FUNCTION_BLOCK FB_Station IMPLEMENTS I_Station
VAR
	refCylinder	: REFERENCE TO FB_Cylinder;
	_eState		: E_StationState;
	_eCommand	: E_Command;
	_stStatus	: ST_StationStatus;
	_stRecipe	: ST_Recipe;
	_uWord		: U_Word;
	_sIdent		: T_Ident;
	_nErrorId	: UDINT;
END_VAR

Cyclic();

METHOD Cyclic
VAR
	bExtended	: BOOL;
END_VAR
bExtended := refCylinder.bIsExtended;

CASE _eState OF
	E_StationState.Idle:
		IF _eCommand = E_Command.Start THEN
			_eState := E_StationState.Running;
		END_IF

	E_StationState.Running:
		IF bExtended THEN
			refCylinder.Retract();
		ELSE
			refCylinder.Extend();
		END_IF
		IF _nErrorId <> 0 THEN
			_eState := E_StationState.Error;
		END_IF

	E_StationState.Error:
		_stStatus.bError := TRUE;

	E_StationState.Done:
		_stStatus.bDone := TRUE;
END_CASE

_stStatus.eState := _eState;
_stStatus.nErrorId := _nErrorId;
_uWord.nWord := _stRecipe.aSteps[1];
END_METHOD

METHOD Execute : BOOL
VAR
END_VAR
IF _eState = E_StationState.Idle THEN
	_eCommand := E_Command.Start;
	_stStatus.bBusy := TRUE;
	Execute := TRUE;
ELSE
	Execute := FALSE;
END_IF
END_METHOD

METHOD Reset : BOOL
VAR
END_VAR
_eState := E_StationState.Idle;
_eCommand := E_Command.None;
_nErrorId := 0;
_stStatus.bBusy := FALSE;
_stStatus.bDone := FALSE;
_stStatus.bError := FALSE;
_stStatus.nErrorId := 0;
Reset := TRUE;
END_METHOD

PROPERTY State : E_StationState
GET
State := _eState;
END_GET
SET
_eState := State;
END_SET
END_PROPERTY

PROPERTY ErrorId : UDINT
GET
ErrorId := _nErrorId;
END_GET
END_PROPERTY

ACTION Act_Home:
refCylinder REF= GVL_System.fbCylinder;
refCylinder.Retract();
_eState := E_StationState.Idle;
_sIdent := 'STATION-01';
END_ACTION

END_FUNCTION_BLOCK

(* stored: Version 1.1.0.1, ProductVersion 3.1.4024.12
   POU FB_Station: Id {ba9b86f0-e4ae-49bd-8d10-d23550802ca5}, SpecialFunc None
   Folder Actions: Id {e81da3d1-8551-49cc-bce9-534df56315e3}
   Method Cyclic: Id {d83d5f63-b782-429a-b4e4-1fd8aac79cdb}
   Method Execute: Id {e043de6a-b3b7-4a09-ac5a-903c66262592}
   Method Reset: Id {ed197d53-3022-4f16-b73a-835f98c1ee8e}
   Property State: Id {0eea66ef-e1f3-405c-94a3-a03642077656}
   Get Get: Id {63d057f4-2d32-45db-b11c-a1f12b0dc2aa}
   Set Set: Id {7a80d7e3-ea77-4397-819a-703c291690f4}
   Property ErrorId: Id {0ad169ae-eccd-45ee-a91a-5754a2bb9e70}
   Get Get: Id {64495b07-7473-4b43-adda-99b867e3bb91}
   Action Act_Home: Id {9d93a169-23da-4f6b-95a9-7d944e47a546} *)
